// TIA Portal V20 export
DATA_BLOCK "BK04"   // DB40116
// stored: MemoryReserve 100
   VAR
      "X10-1 STACK #1 NG CLAMP MOVER OPEN" : Bool;
      "X11-1 STACK #1 NG CLAMP RIGHT OPEN" : Bool;
      "X12-1 STACK #1 NG CLAMP LEFT OPEN" : Bool;
      "X13-1 STAKC #1 NG CLAMP Z-AXIS UP" : Bool;
      "X14-1 STAKC #1 NG CLAMP MOVER BACKWARD" : Bool;
      "X15-1 STACK #1 NG BOX LIFT DOWN" : Bool;
      "X16-1 STACK #1 NG BOX LOCK DOWN" : Bool;
      "X17-1 STACK 1 NG BOX FULL SENSOR" : Bool;
      "X10-2 STACK #1 NG CLAMP MOVER CLOSE" : Bool;
      "X11-2 STACK #1 NG CLAMP RIGHT CLOSE" : Bool;
      "X12-2 STACK #1 NG CLAMP LEFT CLOSE" : Bool;
      "X13-2 STAKC #1 NG CLAMP Z-AXIS DOWN" : Bool;
      "X14-2 STAKC #1 NG CLAMP MOVER FORWARD" : Bool;
      "X15-2 STACK #1 NG BOX LIFT UP" : Bool;
      "X16-2 STACK #1 NG BOX LOCK UP" : Bool;
      "X17-2 SPARE" : Bool;
   END_VAR
BEGIN
END_DATA_BLOCK
